// TIA Portal V18 export
DATA_BLOCK "DELETEw"   // DB58
VERSION : 0.1
// stored: AutoNumber true, DBAccessibleFromOPCUA true, InstanceOfName _spot_iteratorWaitForXray, InstanceOfType FB
"_spot_iteratorWaitForXray"
   // VAR_INPUT
   //    ALLOWED : Bool;
   //    xButtonStartAuto : Bool;
   //    motors_all_arrived : Bool;
   //    XRAY_SHOT_DONE : Bool;
   //    Spot_i_maxN : Int;
   //    sec_siren_done : Real;
   // END_VAR
   // VAR_OUTPUT
   //    reset_PC_SHOT_DONE : Bool;
   //    state_comment : WString;
   //    cycleActive : Bool;
   //    motos_go_now_command : Bool;
   //    XRAY_READYFORSHOT : Bool;
   //    ySirenDone : Bool;
   // END_VAR
   // VAR_IN_OUT
   //    spot_i : Int;
   //    state : UInt;
   // END_VAR
   // VAR
   //    pt_siren_done { ExternalAccessible := 'False'; ExternalVisible := 'False'; ExternalWritable := 'False'} : Time;
   //    mem1 : Bool;
   //    mem2 : Bool;
   //    tons12 { S7_SetPoint := 'True'} : TON_TIME;
   //    tons20 { S7_SetPoint := 'True'} : TON_TIME;
   //    tons10 { S7_SetPoint := 'True'} : TON_TIME;
   //    pt_xray_stuck_in_done { ExternalAccessible := 'False'; ExternalVisible := 'False'; ExternalWritable := 'False'} : Time;
   //    pt_mot_delay : Time;
   //    tons20a { S7_SetPoint := 'True'} : TON_TIME;
   //    tons24 { S7_SetPoint := 'True'} : TON_TIME;
   //    mem3 : Bool;
   // END_VAR
BEGIN
END_DATA_BLOCK
